// TIA Portal V17 export
// export: Created 2025-03-05T08:00:07.8300431Z, ExportSetting WithDefaults, DisplayName Totally Integrated Automation Portal, DisplayVersion V17 Update 8, DisplayName TIA Portal Openness, DisplayVersion V17 Update 8, DisplayName TIA Portal Version Control Interface, DisplayVersion V17, DisplayName SINAMICS Startdrive Advanced, DisplayVersion V17 SP2, DisplayName SINAMICS Startdrive G110M, G120, G120C, G120D, G120P, G115D, DisplayVersion V17 SP2, DisplayName SINAMICS Startdrive G130, G150, S120, S150, SINAMICS MV, S210, DisplayVersion V17 SP2, DisplayName STEP 7 Professional, DisplayVersion V17 Update 8, DisplayName SINUMERIK ONE STEP 7 Toolbox, DisplayVersion V17 Update 12, DisplayName SINUMERIK 840D sl STEP 7 Toolbox, DisplayVersion V17 Update 12, DisplayName STEP 7 Safety, DisplayVersion V17 Update 6, DisplayName WinCC Advanced, DisplayVersion V17 Update 8
DATA_BLOCK "DB2099_MANUAL_LOAD_DMC"   // DB2099
{ S7_Optimized_Access := 'FALSE'; DB_Accessible_From_OPC_UA := 'FALSE' }
VERSION : 0.1
// stored: AutoNumber false, DBAccessibleFromOPCUA false, DBAccessibleFromWebserver true, IsOnlyStoredInLoadMemory false, IsWriteProtectedInAS false
   VAR
      DMC_UNIT_01_HMI : Array[0..99] of Char;   // DMC UNIT 01 IN THE HMI
      DMC_UNIT_02_HMI : Array[0..99] of Char;   // DMC UNIT 02 IN THE HMI
      DMC_STRING_UNIT_01 : String;   // DMC AUX STRING UNIT 01
      DMC_STRING_UNIT_02 : String;   // DMC AUX STRING UNIT 02
      AUX_CNT_INT_UNIT_01 : Int;
      AUX_CNT_INT_UNIT_02 : Int;
      DMC_ARRAY_CHAR_UNIT_01 : Array[0..99] of Char;   // DMC ARRAY UNIT 01
      DMC_ARRAY_CHAR_UNIT_02 : Array[0..99] of Char;   // DMC ARRAY UNIT 02
      MANUAL_LOADING_OR_DRY_PART_LOADED_UNIT_01 : Bool;   // MANUAL LOADING OR DRY CYCLE PART LOADED IN UNIT 01
      MANUAL_LOADING_OR_DRY_PART_LOADED_UNIT_02 : Bool;   // MANUAL LOADING OR DRY CYCLE PART LOADED IN UNIT 02
      MANUAL_LOADING_OR_DRY_PART_UNLOADED_UNIT_01 : Bool;   // MANUAL LOADING OR DRY CYCLE PART UNLOADED IN UNIT 01
      MANUAL_LOADING_OR_DRY_PART_UNLOADED_UNIT_02 : Bool;   // MANUAL LOADING OR DRY CYCLE PART UNLOADED IN UNIT 02
      MANUAL_LOADING_OR_DRY_PART_LOADED_UNIT_01_P : Bool;   // MANUAL LOADING OR DRY CYCLE PART LOADED IN UNIT 01 PULSE
      MANUAL_LOADING_OR_DRY_PART_LOADED_UNIT_02_P : Bool;   // MANUAL LOADING OR DRY CYCLE PART LOADED IN UNIT 02 PULSE
      MANUAL_LOADING_OR_DRY_PART_UNLOADED_UNIT_01_P : Bool;   // MANUAL LOADING OR DRY CYCLE PART UNLOADED IN UNIT 01 PULSE
      MANUAL_LOADING_OR_DRY_PART_UNLOADED_UNIT_02_P : Bool;   // MANUAL LOADING OR DRY CYCLE PART UNLOADED IN UNIT 02 PULSE
      START_DMC_NUMBER_INT : DInt;
      START_DMC_NUMBER_STRING : String;
      START_DMC_NUMBER_CHAR_ARRAY : Array[0..10] of Char;
      AUX_CNT_START_DMC_NUMBER : Int;
      PULSE_1 : Bool;
      PRODUCTION_SELECTED : Bool;
   END_VAR
BEGIN
END_DATA_BLOCK
